FUNCTION detectStabilizedAngle:LREAL
VAR_INPUT
	current_yaw:LREAL;
END_VAR
VAR_OUTPUT
	stab_angle:LREAL;
END_VAR
VAR
END_VAR

IF ((current_yaw >= 0 AND current_yaw <= 45))THEN
      stab_angle := 0;
 	robotdata.robot_direction := 0;
    
	ELSIF ((current_yaw >= 315 AND current_yaw <= 360))THEN
      stab_angle := 360;
	robotdata.robot_direction := 0;
    
    ELSIF ( (current_yaw >= 270 AND current_yaw <= 315)OR (current_yaw >= 225 AND current_yaw <= 270))  THEN
      stab_angle := 270;
     robotdata.robot_direction := 1;
    ELSIF ((current_yaw <= 225 AND current_yaw >= 180)OR(current_yaw >= 135 AND current_yaw <= 180))  THEN
      stab_angle := 180;
     robotdata.robot_direction := 2;
    
    ELSE 
     stab_angle := 90;
	  robotdata.robot_direction := 3;
    END_IF
	detectStabilizedAngle:=stab_angle;

END_FUNCTION

(* stored: Version 1.1.0.1, ProductVersion 3.1.4024.12
   POU detectStabilizedAngle: Id {825e6914-1b47-48e4-b465-321766633e7c}, SpecialFunc None *)
